// Mitsubishi GX Works2 project: A1-60MR-GX2-Ver2   PLC: FX3G

PROGRAM MAIN
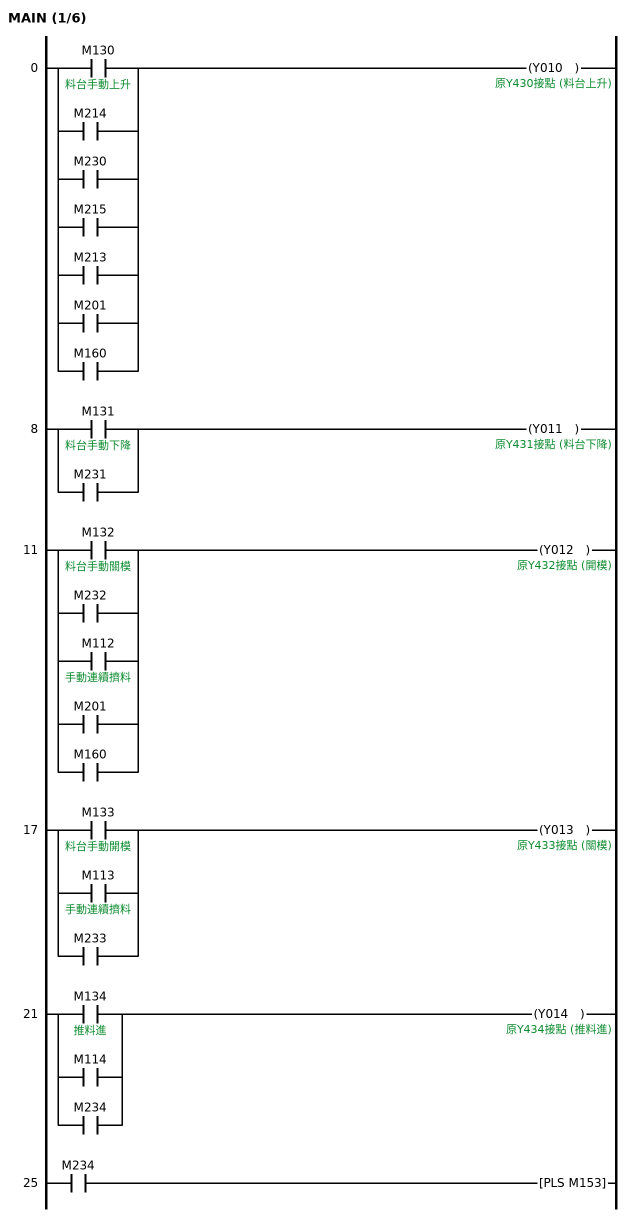
0     LD      M130  ; 料台手動上升
      OR      M214
      OR      M230
      OR      M215
      OR      M213
      OR      M201
      OR      M160
      OUT     Y010  ; 原Y430接點 (料台上升)
8     LD      M131  ; 料台手動下降
      OR      M231
      OUT     Y011  ; 原Y431接點 (料台下降)
11    LD      M132  ; 料台手動關模
      OR      M232
      OR      M112  ; 手動連續擠料
      OR      M201
      OR      M160
      OUT     Y012  ; 原Y432接點 (開模)
17    LD      M133  ; 料台手動開模
      OR      M113  ; 手動連續擠料
      OR      M233
      OUT     Y013  ; 原Y433接點 (關模)
21    LD      M134  ; 推料進
      OR      M114
      OR      M234
      OUT     Y014  ; 原Y434接點 (推料進)
25    LD      M234
      PLS     M153
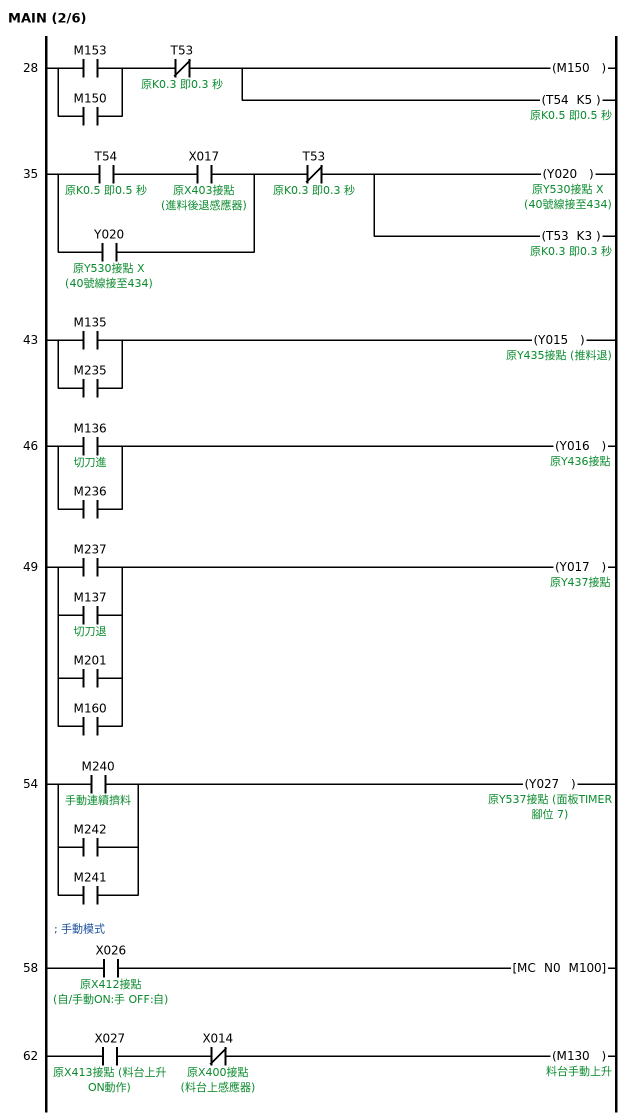
28    LD      M153
      OR      M150
      ANI     T53  ; 原K0.3 即0.3 秒
      OUT     M150
      OUT     T54 K5  ; 原K0.5 即0.5 秒
35    LD      T54  ; 原K0.5 即0.5 秒
      AND     X017  ; 原X403接點 (進料後退感應器)
      OR      Y020  ; 原Y530接點 X (40號線接至434)
      ANI     T53  ; 原K0.3 即0.3 秒
      OUT     Y020  ; 原Y530接點 X (40號線接至434)
      OUT     T53 K3  ; 原K0.3 即0.3 秒
43    LD      M135
      OR      M235
      OUT     Y015  ; 原Y435接點 (推料退)
46    LD      M136  ; 切刀進
      OR      M236
      OUT     Y016  ; 原Y436接點
49    LD      M237
      OR      M137  ; 切刀退
      OR      M201
      OR      M160
      OUT     Y017  ; 原Y437接點
54    LD      M240  ; 手動連續擠料
      OR      M242
      OR      M241
      OUT     Y027  ; 原Y537接點 (面板TIMER 腳位 7)
; 手動模式
58    LD      X026  ; 原X412接點 (自/手動ON:手 OFF:自)
      MC      N0 M100
62    LD      X027  ; 原X413接點 (料台上升 ON動作)
      ANI     X014  ; 原X400接點 (料台上感應器)
      OUT     M130  ; 料台手動上升
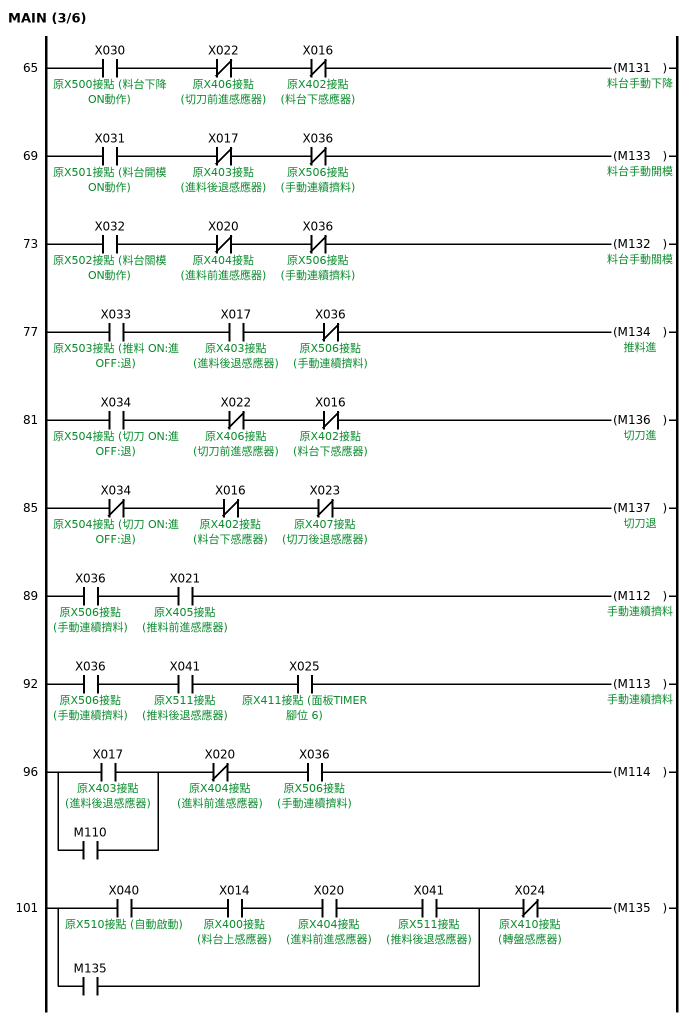
65    LD      X030  ; 原X500接點 (料台下降 ON動作)
      ANI     X022  ; 原X406接點 (切刀前進感應器)
      ANI     X016  ; 原X402接點 (料台下感應器)
      OUT     M131  ; 料台手動下降
69    LD      X031  ; 原X501接點 (料台開模 ON動作)
      ANI     X017  ; 原X403接點 (進料後退感應器)
      ANI     X036  ; 原X506接點 (手動連續擠料)
      OUT     M133  ; 料台手動開模
73    LD      X032  ; 原X502接點 (料台關模 ON動作)
      ANI     X020  ; 原X404接點 (進料前進感應器)
      ANI     X036  ; 原X506接點 (手動連續擠料)
      OUT     M132  ; 料台手動關模
77    LD      X033  ; 原X503接點 (推料 ON:進 OFF:退)
      AND     X017  ; 原X403接點 (進料後退感應器)
      ANI     X036  ; 原X506接點 (手動連續擠料)
      OUT     M134  ; 推料進
81    LD      X034  ; 原X504接點 (切刀 ON:進 OFF:退)
      ANI     X022  ; 原X406接點 (切刀前進感應器)
      ANI     X016  ; 原X402接點 (料台下感應器)
      OUT     M136  ; 切刀進
85    LDI     X034  ; 原X504接點 (切刀 ON:進 OFF:退)
      ANI     X016  ; 原X402接點 (料台下感應器)
      ANI     X023  ; 原X407接點 (切刀後退感應器)
      OUT     M137  ; 切刀退
89    LD      X036  ; 原X506接點 (手動連續擠料)
      AND     X021  ; 原X405接點 (推料前進感應器)
      OUT     M112  ; 手動連續擠料
92    LD      X036  ; 原X506接點 (手動連續擠料)
      AND     X041  ; 原X511接點 (推料後退感應器)
      AND     X025  ; 原X411接點 (面板TIMER 腳位 6)
      OUT     M113  ; 手動連續擠料
96    LD      X017  ; 原X403接點 (進料後退感應器)
      OR      M110
      ANI     X020  ; 原X404接點 (進料前進感應器)
      AND     X036  ; 原X506接點 (手動連續擠料)
      OUT     M114
101   LD      X040  ; 原X510接點 (自動啟動)
      AND     X014  ; 原X400接點 (料台上感應器)
      AND     X020  ; 原X404接點 (進料前進感應器)
      AND     X041  ; 原X511接點 (推料後退感應器)
      OR      M135
      ANI     X024  ; 原X410接點 (轉盤感應器)
      OUT     M135
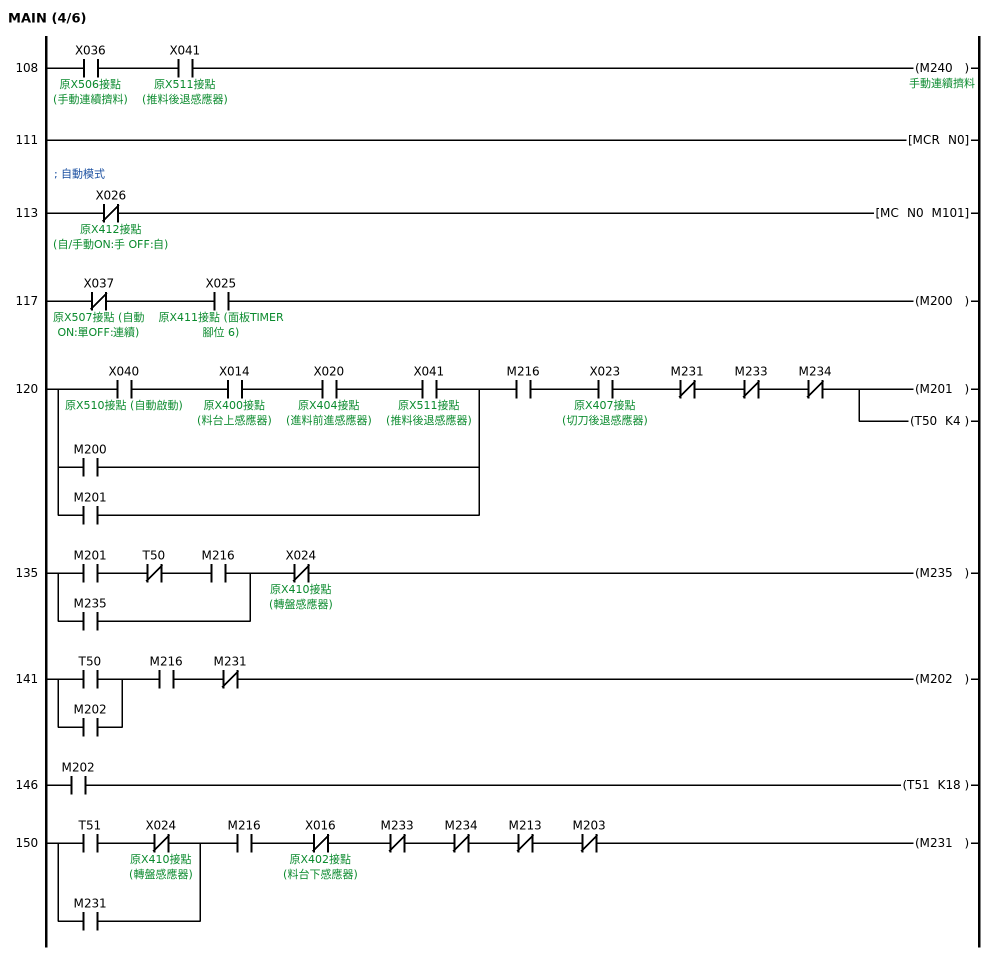
108   LD      X036  ; 原X506接點 (手動連續擠料)
      AND     X041  ; 原X511接點 (推料後退感應器)
      OUT     M240  ; 手動連續擠料
111   MCR     N0
; 自動模式
113   LDI     X026  ; 原X412接點 (自/手動ON:手 OFF:自)
      MC      N0 M101
117   LDI     X037  ; 原X507接點 (自動 ON:單OFF:連續)
      AND     X025  ; 原X411接點 (面板TIMER 腳位 6)
      OUT     M200
120   LD      X040  ; 原X510接點 (自動啟動)
      AND     X014  ; 原X400接點 (料台上感應器)
      AND     X020  ; 原X404接點 (進料前進感應器)
      AND     X041  ; 原X511接點 (推料後退感應器)
      OR      M200
      OR      M201
      AND     M216
      AND     X023  ; 原X407接點 (切刀後退感應器)
      ANI     M231
      ANI     M233
      ANI     M234
      OUT     M201
      OUT     T50 K4
135   LD      M201
      ANI     T50
      AND     M216
      OR      M235
      ANI     X024  ; 原X410接點 (轉盤感應器)
      OUT     M235
141   LD      T50
      OR      M202
      AND     M216
      ANI     M231
      OUT     M202
146   LD      M202
      OUT     T51 K18
150   LD      T51
      ANI     X024  ; 原X410接點 (轉盤感應器)
      OR      M231
      AND     M216
      ANI     X016  ; 原X402接點 (料台下感應器)
      ANI     M233
      ANI     M234
      ANI     M213
      ANI     M203
      OUT     M231
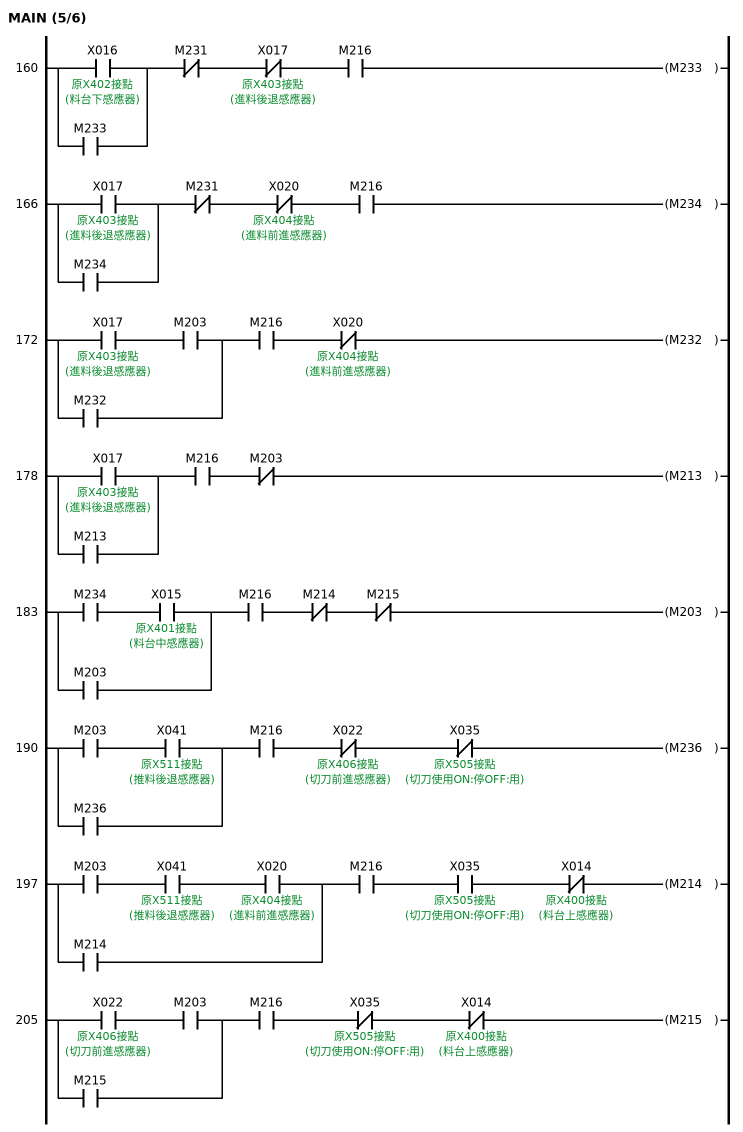
160   LD      X016  ; 原X402接點 (料台下感應器)
      OR      M233
      ANI     M231
      ANI     X017  ; 原X403接點 (進料後退感應器)
      AND     M216
      OUT     M233
166   LD      X017  ; 原X403接點 (進料後退感應器)
      OR      M234
      ANI     M231
      ANI     X020  ; 原X404接點 (進料前進感應器)
      AND     M216
      OUT     M234
172   LD      X017  ; 原X403接點 (進料後退感應器)
      AND     M203
      OR      M232
      AND     M216
      ANI     X020  ; 原X404接點 (進料前進感應器)
      OUT     M232
178   LD      X017  ; 原X403接點 (進料後退感應器)
      OR      M213
      AND     M216
      ANI     M203
      OUT     M213
183   LD      M234
      AND     X015  ; 原X401接點 (料台中感應器)
      OR      M203
      AND     M216
      ANI     M214
      ANI     M215
      OUT     M203
190   LD      M203
      AND     X041  ; 原X511接點 (推料後退感應器)
      OR      M236
      AND     M216
      ANI     X022  ; 原X406接點 (切刀前進感應器)
      ANI     X035  ; 原X505接點 (切刀使用ON:停OFF:用)
      OUT     M236
197   LD      M203
      AND     X041  ; 原X511接點 (推料後退感應器)
      AND     X020  ; 原X404接點 (進料前進感應器)
      OR      M214
      AND     M216
      AND     X035  ; 原X505接點 (切刀使用ON:停OFF:用)
      ANI     X014  ; 原X400接點 (料台上感應器)
      OUT     M214
205   LD      X022  ; 原X406接點 (切刀前進感應器)
      AND     M203
      OR      M215
      AND     M216
      ANI     X035  ; 原X505接點 (切刀使用ON:停OFF:用)
      ANI     X014  ; 原X400接點 (料台上感應器)
      OUT     M215
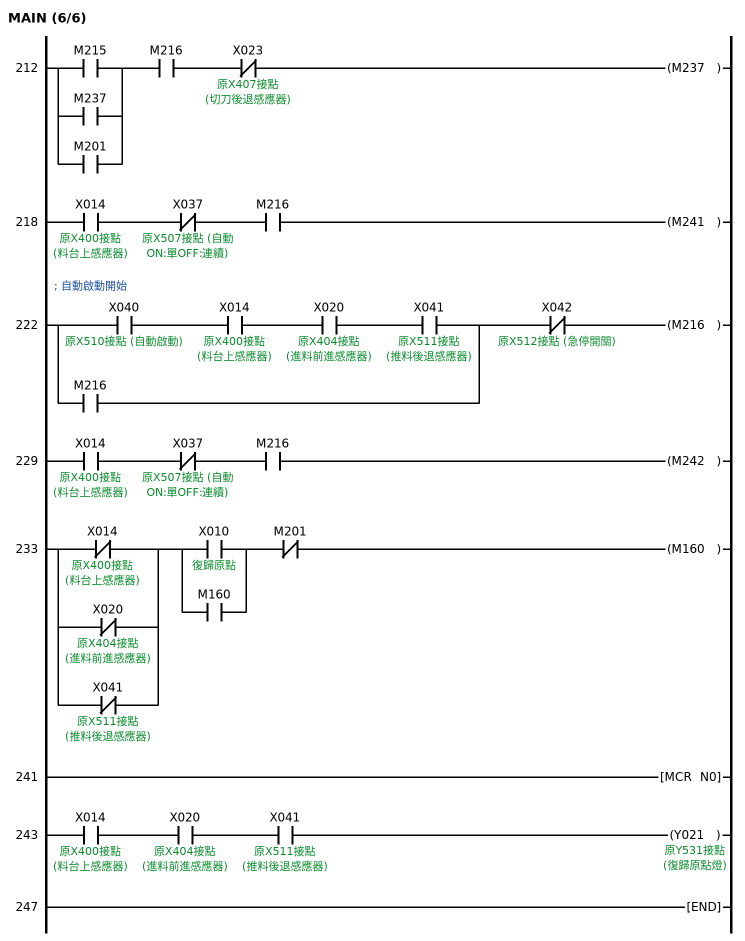
212   LD      M215
      OR      M237
      OR      M201
      AND     M216
      ANI     X023  ; 原X407接點 (切刀後退感應器)
      OUT     M237
218   LD      X014  ; 原X400接點 (料台上感應器)
      ANI     X037  ; 原X507接點 (自動 ON:單OFF:連續)
      AND     M216
      OUT     M241
; 自動啟動開始
222   LD      X040  ; 原X510接點 (自動啟動)
      AND     X014  ; 原X400接點 (料台上感應器)
      AND     X020  ; 原X404接點 (進料前進感應器)
      AND     X041  ; 原X511接點 (推料後退感應器)
      OR      M216
      ANI     X042  ; 原X512接點 (急停開關)
      OUT     M216
229   LD      X014  ; 原X400接點 (料台上感應器)
      ANI     X037  ; 原X507接點 (自動 ON:單OFF:連續)
      AND     M216
      OUT     M242
233   LDI     X014  ; 原X400接點 (料台上感應器)
      ORI     X020  ; 原X404接點 (進料前進感應器)
      ORI     X041  ; 原X511接點 (推料後退感應器)
      LD      X010  ; 復歸原點
      OR      M160
      ANB
      ANI     M201
      OUT     M160
241   MCR     N0
243   LD      X014  ; 原X400接點 (料台上感應器)
      AND     X020  ; 原X404接點 (進料前進感應器)
      AND     X041  ; 原X511接點 (推料後退感應器)
      OUT     Y021  ; 原Y531接點 (復歸原點燈)
247   END
END_PROGRAM

// device comments not shown above
Y022  ; 原Y532接點 X
Y023  ; 原Y533接點 X
Y024  ; 原Y534接點 X
Y025  ; 原Y535接點 X
Y026  ; 原Y536接點 X
X043  ; 原X513接點
